// TIA Portal project "simulation1" (V15)

(* hardware
DEVICE "S7-1200 station_1"  S7-1200 Station
   slot 0: "Rack_0"  S7-1200 Rack  Rack  V1.0
   slot 1: "PLC_1"  CPU 1214C DC/DC/DC  6ES7 214-1AG40-0XB0  V4.2
   slot 3: "AQ 1x12BIT_1"  AQ1 signal board  6ES7 232-4HA30-0XB0  V1.0
   slot 101: "CM 1243-5"  CM 1243-5  6GK7 243-5DX30-0XE0  V1.3
   slot 102: "CM 1241 (RS485)_1"  CM 1241 (RS485)  6ES7 241-1CH30-0XB0  V1.0
*)

// ===== PLC "PLC_1"  CPU 1214C DC/DC/DC =====

VAR_GLOBAL   // PLC tag table "Default tag table"
   ""StartStop"" AT %I0.0 : Bool;
   ""CLewo"" AT %I0.2 : Bool;
   ""CPrawo"" AT %I0.3 : Bool;
   ""krotki"" AT %I0.4 : Bool;
   ""sredni"" AT %I0.5 : Bool;
   ""dlugi"" AT %I0.6 : Bool;
   ""podzielnik"" AT %Q0.0 : Bool;
   ""kLewo"" AT %Q0.1 : Bool;
   ""kPrawo"" AT %Q0.2 : Bool;
   ""wyjscie_krotki"" AT %Q0.4 : Bool;
   ""wyjscie_sredni"" AT %Q0.5 : Bool;
   ""wyjscie_dlugi"" AT %Q0.6 : Bool;
END_VAR